FUNCTION_BLOCK SPLIT_AD_INTO_AX (* this Function splits the 32 AX (BOOL) adapters from a AD (DWORD) *)
  (* Standard: 61499-2; Description: Copyright (c) 2026 Meisterschulen am Ostbahnhof SPDX-License-Identifier: EPL-2.0 *)
  (* Version 1.0, 2026-05-16, Franz Höpfinger, Meisterschulen am Ostbahnhof, initial API and implementation and/or initial documentation *)
  PACKAGE adapter::splitting;
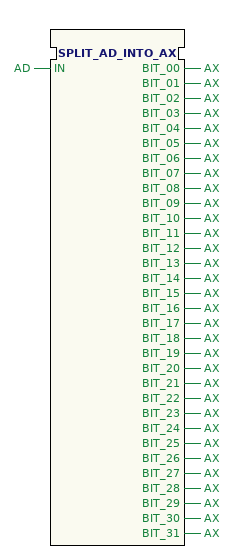
  SOCKETS
    IN : adapter::types::unidirectional::AD; (* DWORD Input *)
  END_SOCKETS
  PLUGS
    BIT_00 : adapter::types::unidirectional::AX; (* Bool Bit 0 *)
    BIT_01 : adapter::types::unidirectional::AX; (* Bool Bit 1 *)
    BIT_02 : adapter::types::unidirectional::AX; (* Bool Bit 2 *)
    BIT_03 : adapter::types::unidirectional::AX; (* Bool Bit 3 *)
    BIT_04 : adapter::types::unidirectional::AX; (* Bool Bit 4 *)
    BIT_05 : adapter::types::unidirectional::AX; (* Bool Bit 5 *)
    BIT_06 : adapter::types::unidirectional::AX; (* Bool Bit 6 *)
    BIT_07 : adapter::types::unidirectional::AX; (* Bool Bit 7 *)
    BIT_08 : adapter::types::unidirectional::AX; (* Bool Bit 8 *)
    BIT_09 : adapter::types::unidirectional::AX; (* Bool Bit 9 *)
    BIT_10 : adapter::types::unidirectional::AX; (* Bool Bit 10 *)
    BIT_11 : adapter::types::unidirectional::AX; (* Bool Bit 11 *)
    BIT_12 : adapter::types::unidirectional::AX; (* Bool Bit 12 *)
    BIT_13 : adapter::types::unidirectional::AX; (* Bool Bit 13 *)
    BIT_14 : adapter::types::unidirectional::AX; (* Bool Bit 14 *)
    BIT_15 : adapter::types::unidirectional::AX; (* Bool Bit 15 *)
    BIT_16 : adapter::types::unidirectional::AX; (* Bool Bit 16 *)
    BIT_17 : adapter::types::unidirectional::AX; (* Bool Bit 17 *)
    BIT_18 : adapter::types::unidirectional::AX; (* Bool Bit 18 *)
    BIT_19 : adapter::types::unidirectional::AX; (* Bool Bit 19 *)
    BIT_20 : adapter::types::unidirectional::AX; (* Bool Bit 20 *)
    BIT_21 : adapter::types::unidirectional::AX; (* Bool Bit 21 *)
    BIT_22 : adapter::types::unidirectional::AX; (* Bool Bit 22 *)
    BIT_23 : adapter::types::unidirectional::AX; (* Bool Bit 23 *)
    BIT_24 : adapter::types::unidirectional::AX; (* Bool Bit 24 *)
    BIT_25 : adapter::types::unidirectional::AX; (* Bool Bit 25 *)
    BIT_26 : adapter::types::unidirectional::AX; (* Bool Bit 26 *)
    BIT_27 : adapter::types::unidirectional::AX; (* Bool Bit 27 *)
    BIT_28 : adapter::types::unidirectional::AX; (* Bool Bit 28 *)
    BIT_29 : adapter::types::unidirectional::AX; (* Bool Bit 29 *)
    BIT_30 : adapter::types::unidirectional::AX; (* Bool Bit 30 *)
    BIT_31 : adapter::types::unidirectional::AX; (* Bool Bit 31 *)
  END_PLUGS
END_FUNCTION_BLOCK
